Staubli VAL3: getFrame.pgx

public program getFrame(frame& x_fFrame[], bool x_bCycle)
  local num l_nIndex
begin
end
